// TwinCAT 3 PLC project Base
// ProgramVersion: 3.1.4022.4
// libraries:
//   Tc2_Standard, * (Beckhoff Automation GmbH)
//   Tc2_System, * (Beckhoff Automation GmbH)
//   Tc2_Utilities, * (Beckhoff Automation GmbH)
//   Tc3_IotBase, * (Beckhoff Automation GmbH)
//   Tc3_IotCommunicator, * (Beckhoff Automation GmbH)
//   Tc3_JsonXml, * (Beckhoff Automation GmbH)
//   Tc3_Module, * (Beckhoff Automation GmbH)
// project tree:
//   DUTs/ E_JsonStates.TcDUT (not stored), ST_ReceivedData.TcDUT
//   GVLs/ CELL_STATE.TcGVL (not stored), CELL_WORKING_STATES.TcGVL, CLAMP_STATE.TcGVL, CELL_ACTION_STATE.TcGVL (not stored), DATA_SERVICE_STATE.TcGVL (not stored), MHS_STATE.TcGVL (not stored), MHS_Registers.TcGVL
//   / PlcTask.TcTTO
//   POUs/ FB_Bool_To_Word.TcPOU (not stored), FB_Cell_Simu.TcPOU, FB_InterfaceProfibus.TcPOU (not stored), FB_RESTapi.TcPOU, FB_VirtualCell.TcPOU (not stored), FB_Word_To_Bool.TcPOU (not stored), I_CELL.TcIO, FB_Cell.TcPOU, FB_Clamp.TcPOU, FB_ClampSimulated.TcPOU, FB_DataService.TcPOU (not stored), FB_InterfaceIO.TcPOU (not stored), FB_InterfaceSimulated.TcPOU, FB_MHS.TcPOU, ITF_Cell.TcIO (not stored), JsonSaxHandler.TcPOU (not stored), MAIN.TcPOU, FB_VirtualCellIntWriter.TcPOU (not stored)
//   POUs/REST/ MAIN_1.TcPOU
//   POUs/REST/Postman/ FB_Get.TcPOU, FB_PUT.TcPOU
// real-time tasks:
//   TASK PlcTask: cycle T#10ms, priority 20, ADS port 350
// I/O:
//   DEVICE Device 3 (EtherCAT) (disabled), AmsNetId 192.168.74.113.4.1
//     Box 1 (CU1128) [CU1128 6x EtherCAT junction]
//       A2_Schaltschrank [EK1100 EtherCAT Coupler (2A E-Bus)]
//         Term 3 (EL2004) [EL2004 4Ch. Dig. Output 24V, 0.5A]
//         Term 4 (EL1004) [EL1004 4Ch. Dig. Input 24V, 3ms]
//         Term 5 (EL2004) [EL2004 4Ch. Dig. Output 24V, 0.5A]
//         Term 6 (EL2004) [EL2004 4Ch. Dig. Output 24V, 0.5A]
//         Term 7 (EL1004) [EL1004 4Ch. Dig. Input 24V, 3ms]
//         Term 8 (EL1004) [EL1004 4Ch. Dig. Input 24V, 3ms]
//         Term 9 (EL2004) [EL2004 4Ch. Dig. Output 24V, 0.5A]
//         Term 10 (EL1004) [EL1004 4Ch. Dig. Input 24V, 3ms]
//         Term 24 (EL9011) [EL9011 End Terminal]
//       A5 [EK1100 EtherCAT Coupler (2A E-Bus)]
//         Term 12 (EL1004) [EL1004 4Ch. Dig. Input 24V, 3ms]
//         Term 13 (EL1004) [EL1004 4Ch. Dig. Input 24V, 3ms]
//         Term 14 (EL2004) [EL2004 4Ch. Dig. Output 24V, 0.5A]
//         Term 15 (EL2004) [EL2004 4Ch. Dig. Output 24V, 0.5A]
//         Term 16 (EL2004) [EL2004 4Ch. Dig. Output 24V, 0.5A]
//         Term 25 (EL9011) [EL9011 End Terminal]
//       Dummy term [CU1128 6x EtherCAT junction - Dev A]
//         Term 18 (EK1100) [EK1100 EtherCAT Coupler (2A E-Bus)]
//           Term 19 (EL1004) [EL1004 4Ch. Dig. Input 24V, 3ms]
//           Term 20 (EL9505) [EL9505 Power supply terminal 5V]
//           Term 21 (EL1124) [EL1124 4Ch. Dig. Input 5V, 10µs, Sensor Power]
//           Term 22 (EL2124) [EL2124 4Ch. Dig. Output 5V, 20mA]
//           Term 26 (EL9011) [EL9011 End Terminal]
//       Term 25 (CU1128-C) [CU1128 6x EtherCAT junction - Dev B]

CONFIGURATION Base
    RESOURCE PLC ON TwinCAT3
        TASK PlcTask(INTERVAL := T#10ms, PRIORITY := 20);
        PROGRAM MAIN_1 WITH PlcTask : MAIN_1;
    END_RESOURCE
END_CONFIGURATION

// ---- DUTs/ST_ReceivedData.TcDUT
TYPE ST_ReceivedData :
STRUCT
	userId:	DINT;
	id:		DINT;
	title:	STRING(255);
	body:	STRING(255);
END_STRUCT
END_TYPE

// ---- GVLs/CELL_WORKING_STATES.TcGVL
{attribute 'qualified_only'}
VAR_GLOBAL
TYPE
	CELL_WORKING_STATES: (e_START, e_WORKING, e_DATAPUT,e_FINISHED);
END_TYPE		

END_VAR

// ---- GVLs/CLAMP_STATE.TcGVL
{attribute 'qualified_only'}
VAR_GLOBAL
TYPE
	CLAMP_STATE: (e_OPEN, e_CLOSED_FULL, e_CLOSED, e_ERROR);
END_TYPE		

END_VAR

// ---- GVLs/MHS_Registers.TcGVL
{attribute 'qualified_only'}
VAR_GLOBAL
 MHS : ARRAY [1..20] OF DINT;
END_VAR

// ---- POUs/I_CELL.TcIO
INTERFACE I_CELL

METHOD GetErrorString : STRING
VAR_INPUT
END_VAR
END_METHOD

METHOD GetName : STRING
VAR_INPUT
END_VAR
END_METHOD

METHOD GetState : INT
VAR_INPUT
END_VAR
END_METHOD

METHOD GetWorkpiece : DINT
VAR_INPUT
END_VAR
END_METHOD

METHOD IsDisassemblyCell : BOOL
VAR_INPUT
END_VAR
END_METHOD

METHOD IsError : BOOL
VAR_INPUT
END_VAR
END_METHOD

METHOD IsIdle : BOOL
VAR_INPUT
END_VAR
END_METHOD

METHOD IsVirtualCell : BOOL
VAR_INPUT
END_VAR
END_METHOD

METHOD RequestActionState : BOOL
VAR_INPUT
	csStateRequest : CELL_ACTION_STATE;
END_VAR
END_METHOD

METHOD RequestWork : BOOL
VAR_INPUT
END_VAR
END_METHOD

METHOD SetDisassemblyCell : BOOL
VAR_INPUT
	bIsDisassemblyCell : BOOL;
END_VAR
END_METHOD

METHOD SetGetDataServiceEnable : BOOL
VAR_INPUT
END_VAR
END_METHOD

METHOD SetName : BOOL
VAR_INPUT
	sName :string ;
END_VAR
END_METHOD

METHOD SetPutDataServiceEnable : BOOL
VAR_INPUT
END_VAR
END_METHOD

METHOD SetVirtualCell : BOOL
VAR_INPUT
END_VAR
END_METHOD

METHOD SetWorkpiece : BOOL
VAR_INPUT
	iWorkpiece : DINT;
	sWorkpieceID : STRING;
END_VAR
END_METHOD

METHOD StateMachine : BOOL
VAR_INPUT
END_VAR
END_METHOD

METHOD StateMachineProfibus : BOOL
VAR_INPUT
END_VAR
END_METHOD

END_INTERFACE

// ---- POUs/REST/MAIN_1.TcPOU
PROGRAM MAIN_1
VAR
	// trigger command execution for Postman-Echo samples
	
	
	fbMHS :  FB_MHS ;
	
	
	
	
END_VAR

fbMHS();

END_PROGRAM

// ---- POUs/FB_MHS.TcPOU
FUNCTION_BLOCK FB_MHS


VAR
	m_csStateRequest : MHS_STATE;
	m_csStateRequestOld : MHS_STATE;
	m_csState : MHS_STATE;
	m_csStateLastCycle : MHS_STATE;
	m_csStateLastAction : MHS_STATE;
	m_Name : STRING;	
	// Von SystemDemonstratorApp kommend
	m_iWorkpiece : DINT; 
	m_iCell : DINT;
	m_iRequest: DINT;
	// Von SystemDemonstratorApp kommend angenommen
	m_iWorkpieceAccepted : DINT; 
	m_iCellAccepted : DINT;
	m_iRequestAccepted: DINT;
	
	// Von PLC kommend 
	m_iMachineFree : DINT;	
	
	
	//Von MiR kommend
	m_iRequestMachineFree : DINT;
	m_iActionTerminated : DINT;	
	
	
	
	// Zustand der Zelle die Beladen oder Entladen werden soll
	m_eCurrentCellState : CELL_ACTION_STATE;
	m_eNeededCellState : CELL_ACTION_STATE;
	m_bNeededCellStatePending : BOOL;
	
	aMHS : ARRAY [1..20] OF DINT; // Interface API-Array
	
	
	m_iSimulationsTimer : DINT;
	
	///////////////////////////////////////////////////////////////////////////
	
	bGet, bPut   	: BOOL;
	

	
	fbClient				:  FB_IotHttpClient :=(sHostName:='jsonplaceholder.typicode.com',
								  	bKeepAlive:=TRUE, tConnectionTimeout:=T#10S);
								
	fbGet						:ARRAY [1..10] OF FB_Get;
	fbPut						:ARRAY [11..20] OF FB_PUT; 
	/////////////////////////////////////////////////////////////////////////////
	//*Hami* String Replace for URi
	
	s_URI : STRING  			:= '/posts/xx';
	i_Register	  				: INT ;
	s_i_Register				: STRING;
	S_Register_URi				: STRING;
	I							: INT ;
	i_I							: INT;
END_VAR

StateMachine();
//FOR i_Register:=1 TO 10  DO
//	i_Register := i_Register + 1;
//	s_i_Register := INT_TO_STRING(i_Register);
//	S_Register_URi := REPLACE(s_URI , s_i_Register , 2 , 8 );
	
//	I := I +1;
	
// END_FOR 

//IF NOT fbClient.bConfigured THEN 
//		fbClient.nHostPort:= 80;
//	END_IF 


/////////////////////////////////////////////////////////////////////////////////////////		

IF fbClient.bConfigured THEN 
		fbGet[1](bSend:=bGet,sURi := '/posts/1', fbClient:=fbClient);
		fbPut[11](bSend:=bPut,sURi := '/posts/1', fbClient:=fbClient);
END_IF

/////////////////////////////////////////////////////////////////////////////////////////		

IF fbClient.bConfigured THEN 
		fbGet[2](bSend:=bGet,sURi := '/posts/2', fbClient:=fbClient);
		fbPut[12](bSend:=bPut,sURi := '/posts/2', fbClient:=fbClient);
END_IF

/////////////////////////////////////////////////////////////////////////////////////////		

IF fbClient.bConfigured THEN 
		fbGet[3](bSend:=bGet,sURi := '/posts/3', fbClient:=fbClient);
		fbPut[13](bSend:=bPut,sURi := '/posts/3', fbClient:=fbClient);
END_IF

/////////////////////////////////////////////////////////////////////////////////////////		

IF fbClient.bConfigured THEN 
		fbGet[4](bSend:=bGet,sURi := '/posts/4', fbClient:=fbClient);
		fbPut[14](bSend:=bPut,sURi := '/posts/4', fbClient:=fbClient);
END_IF
/////////////////////////////////////////////////////////////////////////////////////////		

IF fbClient.bConfigured THEN 
		fbGet[5](bSend:=bGet,sURi := '/posts/5', fbClient:=fbClient);
		fbPut[15](bSend:=bPut,sURi := '/posts/5', fbClient:=fbClient);
END_IF


	fbClient.Execute();
	

	///////////////////////////// init client parameters at startup////////////////////////////////////
	
	

///////////////////////// SET MHS Connection///////////////////////////
// init client parameters at startup

/////////////////////////////////////////////////////////////////////
(*aMHS[1] := fbGet[1].q_iRegister;
aMHS[2] := fbGet[2].q_iRegister;
aMHS[3] := fbGet[3].q_iRegister;
aMHS[4] := fbGet[4].q_iRegister;
aMHS[5] := fbGet[5].q_iRegister;
aMHS[6] := fbGet[6].q_iRegister;
aMHS[7] := fbGet[7].q_iRegister;
aMHS[8] := fbGet[8].q_iRegister;
aMHS[9] := fbGet[9].q_iRegister;
aMHS[10] := fbGet[10].q_iRegister; 
*)

FOR I:=1 TO 10 DO
	aMHS[I] := fbGet[I].q_iRegister;
END_FOR


FOR i_I:=11 TO 20 DO
	fbPut[I].i_iRegister := aMHS[I];
END_FOR

METHOD GetActionFinished : BOOL
VAR_INPUT
END_VAR
IF m_csState = MHS_STATE.e_AKTION_FINISHED THEN
	GetActionFinished := TRUE;
ELSE
	GetActionFinished := FALSE;
END_IF
END_METHOD

METHOD GetCurrentCellForAction : DINT
VAR_INPUT
END_VAR
GetCurrentCellForAction := m_iCellAccepted;
END_METHOD

METHOD GetState : BOOL
VAR_INPUT
END_VAR
END_METHOD

METHOD NeededCellStatePending : BOOL
VAR_INPUT
END_VAR
NeededCellStatePending := m_bNeededCellStatePending;
m_bNeededCellStatePending := FALSE;
END_METHOD

METHOD RequestAction : BOOL
VAR_INPUT
	
	iWorkpiece : DINT; 
	iCell : DINT;
	bRequest : DINT;
END_VAR

m_iWorkpiece :=  iWorkpiece;
m_iCell := iCell;
m_iRequest := bRequest;
END_METHOD

METHOD RequestState : BOOL
VAR_INPUT
END_VAR
END_METHOD

METHOD SendNeededToCell : CELL_ACTION_STATE
VAR_INPUT
END_VAR
SendNeededToCell := m_eNeededCellState;
END_METHOD

METHOD SetClampIsOpen : BOOL
VAR_INPUT
iClampIsOpen : DINT;	

END_VAR
//IF iClampIsOpen > 0 THEN
//	m_iClampIsOpen := 1;
//	m_iClampIsClose := 0;
//ELSE
//	m_iClampIsOpen := 0;
//	m_iClampIsClose := 1;	
//END_IF
END_METHOD

METHOD SetDoorIsOpen : BOOL
VAR_INPUT
	iDoorIsOpen :DINT;
END_VAR
//IF iDoorIsOpen > 0 THEN
//	m_iDoorIsOpen := 1;
//	m_iDoorIsClose := 0;
//ELSE
//	m_iDoorIsOpen := 0;
//	m_iDoorIsClose := 1;	
//END_IF
END_METHOD

METHOD SetMachineFree : BOOL
VAR_INPUT
	iMachineFree:DINT;
END_VAR
m_iMachineFree := iMachineFree;
END_METHOD

METHOD SetStateCurrentMachineForAction : BOOL
VAR_INPUT
	eCurrentCellState :CELL_ACTION_STATE;
END_VAR
m_eCurrentCellState := eCurrentCellState;

SetStateCurrentMachineForAction := TRUE;
END_METHOD


METHOD StateMachine : BOOL
VAR_INPUT
END_VAR

VAR

END_VAR

	// VOM MHS

	//{define Simulated}
	{define MHSConnected}
	
	{IF defined (MHSConnected)}
 	m_iRequestMachineFree   := aMHS[11];
	m_iActionTerminated :=  aMHS[12];
	{END_IF}
	// PLC interne Variablen
	//m_iDoorIsOpen : DINT;	
	//m_iClampIsOpen : DINT;
	//m_iClampIsClose : DINT;	
	//m_iDoorIsClose : DINT;


	
	
CASE m_csState OF

MHS_STATE.e_IDLE: 

	IF m_iWorkpiece > 0 AND m_iCell > 0 AND m_iRequest > 0 THEN
		m_iWorkpieceAccepted := m_iWorkpiece;  
		m_iCellAccepted := m_iCell;
		m_iRequestAccepted:= m_iRequest; 	
	END_IF

	IF m_iWorkpieceAccepted > 0 AND m_iCellAccepted > 0 AND m_iRequestAccepted = 2 THEN
		aMHS[1] := m_iWorkpieceAccepted;
		aMHS[2] := m_iCellAccepted;
		aMHS[3] := m_iRequestAccepted;
		m_iWorkpiece := 0;
 		m_iCell := 0;
		m_iRequest := 0;
		m_csState := MHS_STATE.e_PGO_POS;	
	END_IF
	IF m_iWorkpieceAccepted > 0 AND m_iCellAccepted > 0 AND m_iRequestAccepted = 1 THEN
		aMHS[1] := m_iWorkpieceAccepted;
		aMHS[2] := m_iCellAccepted;
		aMHS[3] := m_iRequestAccepted;
		m_iWorkpiece := 0;
 		m_iCell := 0;
		m_iRequest := 0;
		m_csState := MHS_STATE.e_GGO_POS;	
	END_IF
	// Löschen dieser Anforderung
	m_iRequestAccepted := 0;


// SUBROUTINE WP in Maschine bringen	  
MHS_STATE.e_PGO_POS:
	
 	IF m_iRequestMachineFree > 0 THEN
		m_eNeededCellState := CELL_ACTION_STATE.e_LoadPos;
		m_bNeededCellStatePending := TRUE;
		m_csState := MHS_STATE.e_PWAIT_DOOR;
	END_IF
	

MHS_STATE.e_PWAIT_DOOR:	
  	IF  m_eCurrentCellState = CELL_ACTION_STATE.e_LoadPos THEN
		//aMHS[3] := 0;//m_iRequest;
		m_iMachineFree := 1;
		m_csState := MHS_STATE.e_PWAIT_CLAMP;
	END_IF

MHS_STATE.e_PWAIT_CLAMP:
		m_csState := MHS_STATE.e_PPUT_WP;
	

MHS_STATE.e_PPUT_WP:
		m_csState := MHS_STATE.e_PCLOSE_CLAMP;
		
 MHS_STATE.e_PCLOSE_CLAMP:
			m_csState := MHS_STATE.e_PLEAFE_MACHINE;
	 
MHS_STATE.e_PLEAFE_MACHINE:
 	IF m_iActionTerminated > 0 THEN
		m_csState := MHS_STATE.e_AKTION_FINISHED;
	END_IF	

// SUBROUTINE WP aus Maschine holen	  
MHS_STATE.e_GGO_POS:
 	IF m_iRequestMachineFree > 0 THEN
		m_eNeededCellState := CELL_ACTION_STATE.e_UnLoadPos;
		m_bNeededCellStatePending := TRUE;
		m_csState := MHS_STATE.e_GWAIT_DOOR;
	END_IF

	
MHS_STATE.e_GWAIT_DOOR:
  	IF  m_eCurrentCellState = CELL_ACTION_STATE.e_UnLoadPos THEN
		m_iMachineFree := 1;
		//aMHS[3] := 0;//m_iRequest;
		m_csState := MHS_STATE.e_GWAIT_CLAMP;
	END_IF

MHS_STATE.e_GWAIT_CLAMP:
	//IF m_iClampIsOpen > 0 THEN
		m_csState := MHS_STATE.e_GGET_WP;
	//END_IF
MHS_STATE.e_GGET_WP:
	//IF 	m_iClampCloseRequest > 0 THEN
		m_csState := MHS_STATE.e_GCLOSE_CLAMP;
	//END_IF
 MHS_STATE.e_GCLOSE_CLAMP:
 	//IF m_iClampIsClose > 0 THEN
			m_csState := MHS_STATE.e_GLEAFE_MACHINE;	 
 	//END_IF
MHS_STATE.e_GLEAFE_MACHINE:
	
 	IF m_iActionTerminated > 0 THEN
		aMHS[3] := 0;//m_iRequest;
		m_csState := MHS_STATE.e_AKTION_FINISHED;
	END_IF		

MHS_STATE.e_AKTION_FINISHED:
	m_csState := MHS_STATE.e_IDLE;
	m_iMachineFree := 0;
	
MHS_STATE.e_ERROR:
	
ELSE
	m_csState := MHS_STATE.e_ERROR;
 
END_CASE
{IF defined (MHSConnected)}
aMHS[4] :=  m_iMachineFree; 
{END_IF}
END_METHOD

END_FUNCTION_BLOCK

// ---- POUs/REST/Postman/FB_Get.TcPOU
FUNCTION_BLOCK FB_Get
VAR_INPUT
	bSend				: BOOL;
	sURi : STRING;
	
END_VAR
VAR_IN_OUT
	fbClient			: FB_IotHttpClient;
END_VAR
VAR_OUTPUT
	bBusy				: BOOL;
	bError				: BOOL;
	q_iRegister 		: DINT;
END_VAR
VAR
	fbHeader: FB_IotHttpHeaderFieldMap ;
	fbRequest			: FB_IotHttpRequest;
	fbJson				: FB_JsonDomParser;
	nState				: UDINT;
	RisingEdge			: R_TRIG;
	
	bGetContentResult	: BOOL;
	sContent			: STRING(511);
	
	bGetJsonResult		: BOOL;
	jsonDoc				: SJsonValue;
	jsonVal				: SJsonValue;
	newJSONval : SJsonValue;
	sResultValue		: STRING;
	
	nReqCount			: UDINT;	
	nResCount			: UDINT;
	nValidResCount		: UDINT;
	nErrCount			: UDINT;
	b : BOOL ;
	stReceivedData : ST_ReceivedData ;
	bOnce: BOOL;
	
END_VAR

 IF bOnce THEN
	fbHeader.AddField('Authorization', 'Basic RmVsaXg6OGM2OTc2ZTViNTQxMDQxNWJkZTkwOGJkNGRlZTE1ZGZiMTY3YTljODczZmM0YmI4YTgxZjZmMmFiNDQ4YTkxOA==', FALSE);
	fbHeader.AddField('Accept-Language', 'de_DE' , FALSE);
	bOnce:= FALSE;
END_IF


RisingEdge(CLK:= bSend );
CASE nState OF
0:	
	IF RisingEdge.Q THEN 
		IF fbRequest.SendRequest(sURi:=sURi, fbClient:=fbClient, eRequestType:=ETcIotHttpRequestType.HTTP_GET, 0, 0, 0) THEN	
//IF fbRequest.GetJsonDomContent(sURi := '/posts/1/' , fbClient := fbClient , eRequestType:=ETcIotHttpRequestType.HTTP_GET ,fbJson := fbJson,0) THEN				
			nState:= 1;
			nReqCount:= nReqCount+1;
			bBusy:= TRUE;
			bError:= FALSE;
		END_IF					
	END_IF
1:
	IF NOT fbRequest.bBusy THEN
		bError:= TRUE;
		IF NOT fbRequest.bError THEN
				bGetContentResult:= fbRequest.GetContent(pContent:= ADR(sContent), nContentSize:= SIZEOF(sContent), bSetNullTermination:= TRUE);
			IF fbRequest.nStatusCode >= 200 AND fbRequest.nStatusCode < 300 THEN
				bGetJsonResult:= FALSE;
				jsonDoc:= fbRequest.GetJsonDomContent(fbJson);
				IF jsonDoc <> 0 THEN
					bGetJsonResult:= TRUE;
					IF fbJson.HasMember(jsonDoc, 'id')  THEN
						jsonVal:= fbJson.FindMember(jsonDoc, 'id');
						q_iRegister := fbJson.GetInt(jsonVal);
						IF fbJson.HasMember(jsonVal, 'title')  THEN
							jsonVal:= fbJson.FindMember(jsonVal, 'title');
							nValidResCount:= nValidResCount+1;
							bError:= FALSE;						
							IF fbJson.IsString(jsonVal) THEN							
								sResultValue:= fbJson.GetString(jsonVal);									
							END_IF
						END_IF		
					END_IF
				END_IF							
				nResCount:= nResCount+1;			
			END_IF
		END_IF
		nState:= 0;
		bBusy:= FALSE;
		IF bError THEN
			nErrCount:= nErrCount+1;
		END_IF
	END_IF  	
END_CASE

END_FUNCTION_BLOCK

// ---- POUs/REST/Postman/FB_PUT.TcPOU
FUNCTION_BLOCK FB_PUT
VAR_INPUT
	bSend		: BOOL;
	i_iRegister : DINT ;
	sURi 		: STRING;
END_VAR
VAR_IN_OUT
	fbClient			: FB_IotHttpClient;
END_VAR
VAR_OUTPUT
	bBusy				: BOOL;
	bError				: BOOL;
END_VAR
VAR
	fbRequest			: FB_IotHttpRequest;
	fbHeader			: FB_IotHttpHeaderFieldMap;
	fbJson				: FB_JsonDomParser;
	//fbJson			: FB_JsonDomParser;
	nState				: UDINT;
	RisingEdge			: R_TRIG;

	bGetContentResult	: BOOL;
	sContent			: STRING(511);
	
	bGetJsonResult		: BOOL;
	jsonDoc				: SJsonValue;
	jsonVal				: SJsonValue;
	bResultValue		: BOOL;
	
	nReqCount			: UDINT;	
	nResCount			: UDINT;
	nValidResCount		: UDINT;
	nErrCount			: UDINT;
	bOnce				: BOOL:= TRUE;
	l_sMessage 			: STRING(255) := '{"id":"5","title":"1547mV"}';
	sMessage			: STRING(255);
	JsonStringValue		: SJsonValue;
	s_iRegister 		: STRING ;
	ss_iRegister		: STRING ;
END_VAR

IF bOnce THEN
	fbHeader.AddField('Authorization', 'Basic RmVsaXg6OGM2OTc2ZTViNTQxMDQxNWJkZTkwOGJkNGRlZTE1ZGZiMTY3YTljODczZmM0YmI4YTgxZjZmMmFiNDQ4YTkxOA==', FALSE);
	fbHeader.AddField('Accept-Language', 'de_DE' , FALSE);
	bOnce:= FALSE;
END_IF

/////////////////////////////////////////////////////////////////////////////
s_iRegister := DINT_TO_STRING(i_iRegister);
sMessage := REPLACE(l_sMessage,s_iRegister,1,8);
JsonStringValue := fbJson.ParseDocument(sMessage);

/////////////////////////////////////////////////////////////////////////////
RisingEdge(CLK:= bSend);
CASE nState OF
0:	
	IF RisingEdge.Q THEN 
		IF fbRequest.SendJsonDomRequest(sUri:= sURi , fbClient:=fbClient, eRequestType:=ETcIotHttpRequestType.HTTP_PUT, fbJson := fbJson, fbHeader:=fbHeader) THEN				
			nState:= 1;
			nReqCount:= nReqCount+1;
			bBusy:= TRUE;
			bError:= FALSE;
		END_IF					
	END_IF
1:
	IF NOT fbRequest.bBusy THEN
		bError:= TRUE;
		IF NOT fbRequest.bError THEN				 
			bGetContentResult:= fbRequest.GetContent(pContent:= ADR(sContent), nContentSize:= SIZEOF(sContent), bSetNullTermination:= TRUE);
			IF fbRequest.nStatusCode >= 200 AND fbRequest.nStatusCode < 300 THEN
				bGetJsonResult:= FALSE;
				jsonDoc:= fbRequest.GetJsonDomContent(fbJson);
				IF jsonDoc <> 0 THEN
					bGetJsonResult:= TRUE;
					
					IF fbJson.HasMember(jsonDoc, 'id') THEN
					//IF fbJson.HasMember(jsonDoc, 'authenticated') THEN
					jsonVal:= fbJson.FindMember(jsonDoc, 'id');
						//jsonVal:= fbJson.FindMember(jsonDoc, 'authenticated');
						IF fbJson.IsInt(jsonVal) THEN
						//IF fbJson.IsBool(jsonVal) THEN
						i_iRegister:= fbJson.GetInt(jsonVal);
							//bResultValue:= fbJson.GetBool(jsonVal);
							nValidResCount:= nValidResCount+1;
							bError:= FALSE;						
						END_IF	
					END_IF
				END_IF							
				nResCount:= nResCount+1;			
			END_IF
		END_IF
		nState:= 0;
		bBusy:= FALSE;
		IF bError THEN
			nErrCount:= nErrCount+1;
		END_IF
	END_IF  	
END_CASE

END_FUNCTION_BLOCK

// ---- POUs/FB_Cell_Simu.TcPOU
FUNCTION_BLOCK FB_Cell_Simu IMPLEMENTS I_CELL
VAR_INPUT
	
END_VAR
VAR_OUTPUT
END_VAR
VAR
	m_csStateRequest : CELL_ACTION_STATE;
	m_csStateRequestOld : CELL_ACTION_STATE;
	m_csState : CELL_ACTION_STATE;
	m_csStateLastCycle : CELL_ACTION_STATE;
	m_csStateLastAction : CELL_ACTION_STATE;
	
	
	m_csSRWorkingState : CELL_WORKING_STATES := CELL_WORKING_STATES.e_FINISHED;
	m_csSRWorkingStateLast : CELL_WORKING_STATES := CELL_WORKING_STATES.e_FINISHED;
	// Eigenschaften
	m_sName : STRING;
	m_bIsDisassemblyCell : BOOL;
	
	
	m_iWorkpiece : DINT;
	m_sWorkpieceID : STRING;
	

	m_csCellState : CELL_STATE;
	m_csCellStateLast : CELL_STATE;

	fbInterface : FB_InterfaceSimulated; //nn wenn keine Eingeänge vorhanden sind, nach zeiten wechsel
	fbClamp : FB_Clamp; 
	
	m_sErrorString : STRING;
	
	// DataServices
	
	fbDataServicePut : FB_DataService;
	m_bDataServicePutEnable : BOOL;
	fbDataServiceGet : FB_DataService;
	m_bDataServiceGetEnable : BOOL;
	m_sConfigString : STRING;
	m_sConfigStringEndGet : STRING  := '_Get.exe';
	m_sConfigStringEndPut : STRING  := '_Put.exe';
	m_sDataServiceDir: STRING  := 'C:\Users\\Nübel\Desktop\Sysdem_Nü_Ulitmate\CUTS\';
	m_sDataServiceIP: STRING  := '192.168.74.113.1.1';
	
END_VAR

METHOD GetErrorString : STRING
VAR_INPUT
END_VAR
END_METHOD

METHOD GetName : STRING
VAR_INPUT
END_VAR
GetName := m_sName;
END_METHOD

METHOD PUBLIC GetState : INT
VAR_INPUT
	
END_VAR
GetState := m_csState;
END_METHOD

METHOD GetWorkpiece : DINT
VAR_INPUT
END_VAR
GetWorkpiece := m_iWorkpiece;
END_METHOD

METHOD IsDisassemblyCell : BOOL
VAR_INPUT
END_VAR
IsDisassemblyCell := m_bIsDisassemblyCell;
END_METHOD

METHOD IsError : BOOL
VAR_INPUT
END_VAR
IF m_csCellState = CELL_STATE.e_ERROR THEN
	IsError := TRUE;
END_IF
END_METHOD

METHOD IsIdle : BOOL
VAR_INPUT
END_VAR
IF m_csCellState = CELL_STATE.e_IDEL THEN
	IsIdle := TRUE;
END_IF
END_METHOD

METHOD IsVirtualCell : BOOL
VAR_INPUT
END_VAR
IsVirtualCell :=FALSE;
END_METHOD

METHOD PUBLIC RequestActionState : BOOL
VAR_INPUT
	csStateRequest : CELL_ACTION_STATE;
END_VAR
m_csStateRequest := csStateRequest;
END_METHOD

METHOD RequestWork : BOOL
VAR_INPUT
END_VAR
m_csCellState := CELL_STATE.e_WORKING;
END_METHOD

METHOD SetDisassemblyCell : BOOL
VAR_INPUT
	bIsDisassemblyCell : BOOL;
END_VAR
m_bIsDisassemblyCell := bIsDisassemblyCell;
END_METHOD

METHOD SetGetDataServiceEnable : BOOL
VAR_INPUT
END_VAR
m_bDataServiceGetEnable := TRUE;
SetGetDataServiceEnable := TRUE;
END_METHOD

METHOD SetName : BOOL
VAR_INPUT
	sName :string ;
END_VAR
m_sName := sName;
END_METHOD

METHOD SetPutDataServiceEnable : BOOL
VAR_INPUT
END_VAR
m_bDataServicePutEnable := TRUE;
SetPutDataServiceEnable := TRUE;
END_METHOD

METHOD SetVirtualCell : BOOL
VAR_INPUT
END_VAR
END_METHOD

METHOD SetWorkpiece : BOOL
VAR_INPUT
	iWorkpiece : DINT;
	sWorkpieceID : STRING;
END_VAR
m_iWorkpiece := iWorkpiece;
m_sWorkpieceID := sWorkpieceID;
END_METHOD

METHOD PUBLIC StateMachine : BOOL
VAR_INPUT
END_VAR

fbInterface();
fbClamp();



// Error-Abfragen
IF fbClamp.IsError() THEN
	m_csCellState := CELL_STATE.e_ERROR; 
	m_sErrorString := 'CLAMP-Error: Clamp is closed without Workpiece';
END_IF


//Zellen Zustandsmaschine

CASE m_csCellState OF 
	CELL_STATE.e_IDEL:
		fbClamp.SetOpenClamp();	
	
		;
 	CELL_STATE.e_MHS_ACTION;
		//SubRoutine für Aktion beim beladen aktuell leer da alles vom MHS gesteuert wird 
	
		;
	CELL_STATE.e_WORKING:
		//SubRoutine zum Durchführen einer Bearbeitung
		
		IF NOT (m_csCellStateLast = m_csCellState) THEN
			m_csSRWorkingState := CELL_WORKING_STATES.e_START;
			IF m_bDataServiceGetEnable THEN
				fbDataServiceGet.SetNetIP('192.168.74.113.1.1');
				fbDataServiceGet.SetWorkingDirectory('C:\Users\Nübel\Desktop\Sysdem_Nü_Ulitmate\CUTS');
				m_sConfigString := 'C:\Users\Nübel\Desktop\Sysdem_Nü_Ulitmate\CUTS\';
				m_sConfigString := CONCAT(m_sConfigString , m_sName); // erstellen des Pfades der Applikation 
				m_sConfigString := CONCAT(m_sConfigString , m_sConfigStringEndGet);
				fbDataServiceGet.SetCommandLine(m_sWorkpieceID);
				fbDataServiceGet.SetPathOfApplication(m_sConfigString);
				fbDataServiceGet.StartDataService();
			END_IF
		END_IF
			
		CASE m_csSRWorkingState OF
			
			CELL_WORKING_STATES.e_START:
				
				IF NOT (m_csSRWorkingStateLast = m_csSRWorkingState )THEN
					m_csStateRequest := CELL_ACTION_STATE.e_Startabel;
				END_IF
				//m_csSRWorkingState:= CELL_WORKING_STATES.e_FINISHED;
				
				IF m_csState = CELL_ACTION_STATE.e_Startabel AND (fbDataServiceGet.IsFinished() OR NOT(m_bDataServiceGetEnable) )  THEN // Zelle bereit zum Starten und DataServiceGet fertig oder nicht konfiguriert
					m_csSRWorkingState:= CELL_WORKING_STATES.e_WORKING;
					fbDataServiceGet.SetIdle();
					m_csStateRequest:= CELL_ACTION_STATE.e_Running;
				END_IF
				
				
			CELL_WORKING_STATES.e_WORKING:
				IF NOT (m_csSRWorkingStateLast = m_csSRWorkingState) THEN
					m_csStateRequest := CELL_ACTION_STATE.e_Running;
				END_IF
				
				IF m_csState = CELL_ACTION_STATE.e_Finished THEN
					m_csSRWorkingState := CELL_WORKING_STATES.e_FINISHED;
					IF m_bDataServicePutEnable THEN
						fbDataServicePut.SetNetIP('192.168.74.113.1.1');
						fbDataServicePut.SetWorkingDirectory('C:\Users\Nübel\Desktop\Sysdem_Nü_Ulitmate\CUTS');
						m_sConfigString := 'C:\Users\Nübel\Desktop\Sysdem_Nü_Ulitmate\CUTS\';						
						m_sConfigString := CONCAT(m_sConfigString , m_sName); // erstellen des Pfades der Applikation 
						m_sConfigString := CONCAT(m_sConfigString , m_sConfigStringEndPut);// erstellen des Pfades der Applikation
						fbDataServicePut.SetCommandLine(m_sWorkpieceID);
						fbDataServicePut.SetPathOfApplication(m_sConfigString);
						fbDataServicePut.StartDataService();
						m_csSRWorkingState := e_DATAPUT;
					END_IF
		
				END_IF
			CELL_WORKING_STATES.e_DATAPUT:
				
					IF fbDataServicePut.IsFinished() THEN
						fbDataServicePut.SetIdle();
						m_csSRWorkingState := CELL_WORKING_STATES.e_FINISHED;
					END_IF
					
					IF fbDataServicePut.IsError() THEN
						fbDataServicePut.SetIdle();
						m_csSRWorkingState := CELL_STATE.e_ERROR;
					END_IF
					
			CELL_WORKING_STATES.e_FINISHED:
				m_csCellState := CELL_STATE.e_IDEL;
			
		END_CASE		
		
	CELL_STATE.e_ERROR:
		m_csState :=CELL_ACTION_STATE.e_ToEmergencyStop;
	
		
END_CASE
m_csSRWorkingStateLast := m_csSRWorkingState;
m_csCellStateLast := m_csCellState;

IF NOT (m_csStateRequestOld = m_csStateRequest) THEN
	m_csState := m_csStateRequest - 1;
	m_csStateRequestOld := m_csStateRequest;
END_IF


// Aktions Zustandsmaschine
CASE m_csState OF 
	CELL_ACTION_STATE.e_ToStandby:
		IF NOT (m_csStateLastCycle = m_csState) THEN
			fbInterface.SetStandby(TRUE);
			m_csStateLastAction := m_csStateLastCycle;
		END_IF
		
		IF fbInterface.GetStandby() THEN
			m_csState := e_Standby; 
		END_IF
		
	CELL_ACTION_STATE.e_Standby :
	
		IF NOT (m_csStateLastCycle = m_csState) THEN
			m_csStateLastAction := m_csStateLastCycle;
		END_IF
		fbInterface.SetStandby(FALSE);
		
	CELL_ACTION_STATE.e_ToLoadPos:
	
		IF NOT (m_csStateLastCycle = m_csState) THEN
			m_csStateLastAction := m_csStateLastCycle;
			fbInterface.SetMoveToLoad(TRUE);
			fbClamp.SetOpenClamp();
		END_IF
		
		IF fbInterface.GetLoadPos() AND fbClamp.IsOpen() THEN
			m_csState := e_LoadPos; 
		END_IF
		
		
	CELL_ACTION_STATE.e_LoadPos:
	
		IF NOT (m_csStateLastCycle = m_csState) THEN
			m_csStateLastAction := m_csStateLastCycle;
		END_IF
		fbInterface.SetMoveToLoad(FALSE);
				
		
	CELL_ACTION_STATE.e_ToStartabel:
	
		IF NOT (m_csStateLastCycle = m_csState) THEN
			m_csStateLastAction := m_csStateLastCycle;
			fbClamp.SetCloseClampFull();
		END_IF
		
		
		IF  fbClamp.IsClosedFull() THEN
			m_csState := e_Startabel; 
		END_IF
		
	CELL_ACTION_STATE.e_Startabel:
	
		IF NOT (m_csStateLastCycle = m_csState) THEN
			m_csStateLastAction := m_csStateLastCycle;
			
		END_IF
		
	CELL_ACTION_STATE.e_ToRunning:
	
		IF NOT (m_csStateLastCycle = m_csState) THEN
			m_csStateLastAction := m_csStateLastCycle;
			fbInterface.SetStart(TRUE);
		END_IF
		
		IF fbInterface.GetIsRunning() THEN
			m_csState := CELL_ACTION_STATE.e_Running; 
		END_IF
		
	CELL_ACTION_STATE.e_Running:
	
		IF NOT (m_csStateLastCycle = m_csState) THEN
			m_csStateLastAction := m_csStateLastCycle;
		END_IF
		fbInterface.SetStart(FALSE);
		IF fbInterface.GetFinished() THEN
			m_csState := CELL_ACTION_STATE.e_Finished;		
		END_IF
	CELL_ACTION_STATE.e_Finished:
		IF NOT (m_csStateLastCycle = m_csState) THEN
			m_csStateLastAction := m_csStateLastCycle;
		END_IF
		
	CELL_ACTION_STATE.e_ToUnLoadPos:
 
		IF NOT (m_csStateLastCycle = m_csState) THEN
			m_csStateLastAction := m_csStateLastCycle;
			fbClamp.SetOpenClamp();
			fbInterface.SetMoveToUnload(TRUE);
			
		END_IF
		
		
		IF fbInterface.GetUnloadPos() AND fbClamp.IsOpen() THEN
			m_csState := e_UnLoadPos; 
			fbInterface.SetMoveToUnload(FALSE);
		END_IF
		
	CELL_ACTION_STATE.e_UnLoadPos:
	
		IF NOT (m_csStateLastCycle = m_csState) THEN
			m_csStateLastAction := m_csStateLastCycle;
		END_IF
		
	CELL_ACTION_STATE.e_ToEmergencyStop:
	
		IF NOT (m_csStateLastCycle = m_csState) THEN
			m_csStateLastAction := m_csStateLastCycle;
		END_IF
		
		
		IF fbInterface.GetEmergencyStop() THEN
			m_csState := e_EmergencyStop; 
		END_IF
		
	CELL_ACTION_STATE.e_EmergencyStop:
	
		IF NOT (m_csStateLastCycle = m_csState) THEN
			m_csStateLastAction := m_csStateLastCycle;
		END_IF
		
	CELL_ACTION_STATE.e_ToEmergencyOff:
	
		IF NOT (m_csStateLastCycle = m_csState) THEN
			m_csStateLastAction := m_csStateLastCycle;
		END_IF
		
		
		IF fbInterface.GetEmergencyStop() THEN
			m_csState := e_EmergencyOff; 
		END_IF
		
	CELL_ACTION_STATE.e_EmergencyOff:
	
		IF NOT (m_csStateLastCycle = m_csState) THEN
			m_csStateLastAction := m_csStateLastCycle;
		END_IF
		
	ELSE
		IF NOT (m_csStateLastCycle = m_csState) THEN
			m_csStateLastAction := m_csStateLastCycle;
		END_IF
		
END_CASE

IF m_bDataServiceGetEnable THEN
	fbDataServiceGet();
END_IF
IF m_bDataServicePutEnable THEN	
	fbDataServicePut();
END_IF

m_csStateLastCycle := m_csState;
END_METHOD

METHOD StateMachineProfibus : BOOL
VAR_INPUT
END_VAR
END_METHOD

END_FUNCTION_BLOCK

// ---- POUs/FB_InterfaceSimulated.TcPOU
FUNCTION_BLOCK FB_InterfaceSimulated IMPLEMENTS ITF_Cell
VAR_INPUT
END_VAR
VAR_OUTPUT
END_VAR
VAR
	 iTimer : INT;
	 iWaitingTime : INT := 500;
END_VAR

METHOD GetEmergencyOff : BOOL
VAR_INPUT
END_VAR

iTimer := iTimer +1;

IF iTimer > iWaitingTime THEN
	GetEmergencyOff := TRUE;
	iTimer := 0;	
END_IF
END_METHOD

METHOD GetEmergencyStop : BOOL
VAR_INPUT
END_VAR

iTimer := iTimer +1;

IF iTimer > iWaitingTime THEN
	GetEmergencyStop := TRUE;
	iTimer := 0;	
END_IF
END_METHOD

METHOD GetFinished : BOOL
VAR_INPUT
END_VAR

iTimer := iTimer +1;

IF iTimer > iWaitingTime THEN
	GetFinished := TRUE;
	iTimer := 0;	
END_IF
END_METHOD

METHOD GetIsRunning : BOOL
VAR_INPUT
END_VAR


iTimer := iTimer +1;

IF iTimer > iWaitingTime THEN
	GetIsRunning := TRUE;
	iTimer := 0;	
END_IF
END_METHOD

METHOD GetLoadPos : BOOL
VAR_INPUT
END_VAR


iTimer := iTimer +1;

IF iTimer > iWaitingTime THEN
	GetLoadPos := TRUE;
	iTimer := 0;	
END_IF
END_METHOD

METHOD GetStandby : BOOL
VAR_INPUT
END_VAR


iTimer := iTimer +1;

IF iTimer > iWaitingTime THEN
	GetStandby := TRUE;
	iTimer := 0;	
END_IF
END_METHOD

METHOD GetStartable : BOOL
VAR_INPUT
END_VAR



iTimer := iTimer +1;

IF iTimer > iWaitingTime THEN
	GetStartable := TRUE;
	iTimer := 0;	
END_IF
END_METHOD

METHOD GetUnloadPos : BOOL
VAR_INPUT
END_VAR


iTimer := iTimer +1;

IF iTimer > iWaitingTime THEN
	GetUnloadPos := TRUE;
	iTimer := 0;	
END_IF
END_METHOD

METHOD SetEmergencyOff : BOOL
VAR_INPUT
	b:BOOL;
END_VAR
END_METHOD

METHOD SetEmergencyStop : BOOL
VAR_INPUT
	b:BOOL;
END_VAR
END_METHOD

METHOD SetLoadPlace : BOOL
VAR_INPUT
	b :BOOL;
END_VAR
END_METHOD

METHOD SetMoveToLoad : BOOL
VAR_INPUT
	b:BOOL;
END_VAR
END_METHOD

METHOD SetMoveToUnload : BOOL
VAR_INPUT
	b:BOOL;
END_VAR
END_METHOD

METHOD SetStandby : BOOL
VAR_INPUT
	b:BOOL;
END_VAR
END_METHOD

METHOD SetStart : BOOL
VAR_INPUT
	b:BOOL;
END_VAR
END_METHOD

END_FUNCTION_BLOCK

// ---- POUs/FB_Clamp.TcPOU
FUNCTION_BLOCK FB_Clamp
VAR_INPUT
	
END_VAR
VAR_OUTPUT
END_VAR
VAR
m_csState : CLAMP_STATE;	
m_csStateRequested : CLAMP_STATE;

//Eingänge
m_bIsOpen AT %I* : BOOL;
m_bIsClosed AT %I* : BOOL;
m_bIsFull AT %I* : BOOL;

//Ausgänge
m_bOpen AT %Q* :BOOL;


END_VAR


StateMachine();

METHOD IsClosed : BOOL
VAR_INPUT
END_VAR
IF m_csState = CLAMP_STATE.e_CLOSED THEN
	IsClosed := TRUE;
END_IF
END_METHOD

METHOD IsClosedFull : BOOL
VAR_INPUT
END_VAR
IF m_csState = CLAMP_STATE.e_CLOSED_FULL THEN
	IsClosedFull := TRUE;
END_IF
END_METHOD

METHOD IsError : BOOL
VAR_INPUT
END_VAR
IF m_csState = CLAMP_STATE.e_ERROR THEN
	IsError := TRUE;
END_IF
END_METHOD

METHOD IsOpen : BOOL
VAR_INPUT
END_VAR
IF m_csState = CLAMP_STATE.e_OPEN THEN
	IsOpen := TRUE;
END_IF
END_METHOD

METHOD SetCloseClampEmpty : BOOL
VAR_INPUT
END_VAR
m_csStateRequested := CLAMP_STATE.e_CLOSED;
m_bOpen := FALSE;
SetCloseClampEmpty:=TRUE;
END_METHOD

METHOD SetCloseClampFull : BOOL
VAR_INPUT
END_VAR
m_csStateRequested := CLAMP_STATE.e_CLOSED_FULL;
m_bOpen := FALSE;
SetCloseClampFull := TRUE;
END_METHOD

METHOD SetOpenClamp : BOOL
VAR_INPUT
END_VAR
m_bOpen := TRUE;
END_METHOD

METHOD StateMachine : BOOL
VAR_INPUT
END_VAR

//m_bIsOpen : BOOL;
//m_bIsClosed : BOOL;
//m_bIsClosedFull : BOOL;

CASE m_csState  OF
	
	CLAMP_STATE.e_OPEN:	

		IF m_bIsClosed THEN
			IF 	m_bIsFull THEN
				m_csState := CLAMP_STATE.e_CLOSED_FULL;		
			ELSE
				m_csState := CLAMP_STATE.e_CLOSED;		
			END_IF 
		
		END_IF
		
		
 	CLAMP_STATE.e_CLOSED_FULL:
	// Fehler wenn falscher Zustand
 		IF m_csStateRequested = CLAMP_STATE.e_CLOSED THEN
  			m_csState := CLAMP_STATE.e_ERROR;
		END_IF
		
		
		IF m_bIsOpen THEN
			m_csState := CLAMP_STATE.e_OPEN;		
		END_IF
	
	CLAMP_STATE.e_CLOSED:
			// Fehler wenn falscher Zustand in diesem Fall: Werkstück erwartet aber nicht im Halter
 		IF m_csStateRequested = CLAMP_STATE.e_CLOSED_FULL THEN
  			m_csState := CLAMP_STATE.e_ERROR;
		END_IF
	
		IF m_bIsOpen THEN
			m_csState := CLAMP_STATE.e_OPEN;		
		END_IF
		
CLAMP_STATE.e_ERROR:
		
END_CASE
END_METHOD

END_FUNCTION_BLOCK

// ---- POUs/FB_RESTapi.TcPOU
FUNCTION_BLOCK FB_RESTapi
VAR_INPUT
END_VAR
VAR_OUTPUT
END_VAR
VAR
	fbREST : 
END_VAR

END_FUNCTION_BLOCK

// ---- POUs/FB_Cell.TcPOU
FUNCTION_BLOCK FB_Cell IMPLEMENTS I_CELL
VAR_INPUT
	
END_VAR
VAR_OUTPUT
END_VAR
VAR
	m_csStateRequest : CELL_ACTION_STATE;
	m_csStateRequestOld : CELL_ACTION_STATE;
	m_csState : CELL_ACTION_STATE;
	m_csStateLastCycle : CELL_ACTION_STATE;
	m_csStateLastAction : CELL_ACTION_STATE;
	
	
	m_csSRWorkingState : CELL_WORKING_STATES := CELL_WORKING_STATES.e_FINISHED;
	m_csSRWorkingStateLast : CELL_WORKING_STATES := CELL_WORKING_STATES.e_FINISHED;
	// Eigenschaften
	m_sName : STRING;
	m_bIsDisassemblyCell : BOOL;
	
	
	m_iWorkpiece : DINT;
	m_sWorkpieceID : STRING;
	

	m_csCellState : CELL_STATE;
	m_csCellStateLast : CELL_STATE;

	fbInterface : FB_InterfaceIO;
	//*Hami* Deklration von FB_InterfaceProfibus (Die Wurde in Method (StateMachine)) aufgerufen
	fbInterfaceProfibus : FB_InterfaceProfibus;
	fbClamp : FB_Clamp; 
	
	m_sErrorString : STRING;
	
	// DataServices
	
	fbDataServicePut : FB_DataService;
	m_bDataServicePutEnable : BOOL;
	fbDataServiceGet : FB_DataService;
	m_bDataServiceGetEnable : BOOL;
	m_sConfigString : STRING;
	m_sConfigStringEndGet : STRING  := '_Get.exe';
	m_sConfigStringEndPut : STRING  := '_Put.exe';

	m_sDataServiceDir: STRING  := 'C:\Users\\Nübel\Desktop\Sysdem_Nü_Ulitmate\CUTS\';
	m_sDataServiceIP: STRING  := '192.168.74.113.1.1';
	

	
	
END_VAR

METHOD GetErrorString : STRING
VAR_INPUT
END_VAR
END_METHOD

METHOD GetName : STRING
VAR_INPUT
END_VAR
GetName := m_sName;
END_METHOD

METHOD PUBLIC GetState : INT
VAR_INPUT
	
END_VAR
GetState := m_csState;
END_METHOD

METHOD GetWorkpiece : DINT
VAR_INPUT
END_VAR
GetWorkpiece := m_iWorkpiece;
END_METHOD

METHOD IsDisassemblyCell : BOOL
VAR_INPUT
END_VAR
IsDisassemblyCell := m_bIsDisassemblyCell;
END_METHOD

METHOD IsError : BOOL
VAR_INPUT
END_VAR
IF m_csCellState = CELL_STATE.e_ERROR THEN
	IsError := TRUE;
END_IF
END_METHOD

METHOD IsIdle : BOOL
VAR_INPUT
END_VAR
IF m_csCellState = CELL_STATE.e_IDEL THEN
	IsIdle := TRUE;
END_IF
END_METHOD

METHOD IsVirtualCell : BOOL
VAR_INPUT
END_VAR
IsVirtualCell :=FALSE;
END_METHOD

METHOD PUBLIC RequestActionState : BOOL
VAR_INPUT
	csStateRequest : CELL_ACTION_STATE;
END_VAR
m_csStateRequest := csStateRequest;
END_METHOD

METHOD RequestWork : BOOL
VAR_INPUT
END_VAR
m_csCellState := CELL_STATE.e_WORKING;
END_METHOD

METHOD SetDisassemblyCell : BOOL
VAR_INPUT
	bIsDisassemblyCell : BOOL;
END_VAR
m_bIsDisassemblyCell := bIsDisassemblyCell;
END_METHOD

METHOD SetGetDataServiceEnable : BOOL
VAR_INPUT
END_VAR
m_bDataServiceGetEnable := TRUE;
SetGetDataServiceEnable := TRUE;
END_METHOD

METHOD SetName : BOOL
VAR_INPUT
	sName :string ;
END_VAR
m_sName := sName;
END_METHOD

METHOD SetPutDataServiceEnable : BOOL
VAR_INPUT
END_VAR
m_bDataServicePutEnable := TRUE;
SetPutDataServiceEnable := TRUE;
END_METHOD

METHOD SetVirtualCell : BOOL
VAR_INPUT
END_VAR
END_METHOD

METHOD SetWorkpiece : BOOL
VAR_INPUT
	iWorkpiece : DINT;
	sWorkpieceID : STRING;
END_VAR
m_iWorkpiece := iWorkpiece;
m_sWorkpieceID := sWorkpieceID;
END_METHOD

METHOD PUBLIC StateMachine : BOOL
VAR_INPUT
END_VAR




fbInterface();
fbClamp();



// Error-Abfragen
IF fbClamp.IsError() THEN
	m_csCellState := CELL_STATE.e_ERROR; 
	m_sErrorString := 'CLAMP-Error: Clamp is closed without Workpiece';
END_IF


//Zellen Zustandsmaschine

CASE m_csCellState OF 
	CELL_STATE.e_IDEL:
		fbClamp.SetOpenClamp();	
	
		;
 	CELL_STATE.e_MHS_ACTION;
		//SubRoutine für Aktion beim beladen aktuell leer da alles vom MHS gesteuert wird 
	
		;
	CELL_STATE.e_WORKING:
		//SubRoutine zum Durchführen einer Bearbeitung
		
		IF NOT (m_csCellStateLast = m_csCellState) THEN
			m_csSRWorkingState := CELL_WORKING_STATES.e_START;
			IF m_bDataServiceGetEnable THEN
				fbDataServiceGet.SetNetIP('192.168.74.113.1.1');
				fbDataServiceGet.SetWorkingDirectory('C:\Users\Nübel\Desktop\Sysdem_Nü_Ulitmate\CUTS');
				m_sConfigString := 'C:\Users\Nübel\Desktop\Sysdem_Nü_Ulitmate\CUTS\';
				m_sConfigString := CONCAT(m_sConfigString , m_sName); // erstellen des Pfades der Applikation 
				m_sConfigString := CONCAT(m_sConfigString , m_sConfigStringEndGet);
				fbDataServiceGet.SetCommandLine(m_sWorkpieceID);
				fbDataServiceGet.SetPathOfApplication(m_sConfigString);
				fbDataServiceGet.StartDataService();
			END_IF
		END_IF
			
		CASE m_csSRWorkingState OF
			
			CELL_WORKING_STATES.e_START:
				
				IF NOT (m_csSRWorkingStateLast = m_csSRWorkingState )THEN
					m_csStateRequest := CELL_ACTION_STATE.e_Startabel;
				END_IF
				//m_csSRWorkingState:= CELL_WORKING_STATES.e_FINISHED;
				
				IF m_csState = CELL_ACTION_STATE.e_Startabel AND (fbDataServiceGet.IsFinished() OR NOT(m_bDataServiceGetEnable) )  THEN // Zelle bereit zum Starten und DataServiceGet fertig oder nicht konfiguriert
					m_csSRWorkingState:= CELL_WORKING_STATES.e_WORKING;
					fbDataServiceGet.SetIdle();
					m_csStateRequest:= CELL_ACTION_STATE.e_Running;
				END_IF
				
				
			CELL_WORKING_STATES.e_WORKING:
				IF NOT (m_csSRWorkingStateLast = m_csSRWorkingState) THEN
					m_csStateRequest := CELL_ACTION_STATE.e_Running;
				END_IF
				
				IF m_csState = CELL_ACTION_STATE.e_Finished THEN
					m_csSRWorkingState := CELL_WORKING_STATES.e_FINISHED;
					IF m_bDataServicePutEnable THEN
						fbDataServicePut.SetNetIP('192.168.74.113.1.1');
						fbDataServicePut.SetWorkingDirectory('C:\Users\Nübel\Desktop\Sysdem_Nü_Ulitmate\CUTS');
						m_sConfigString := 'C:\Users\Nübel\Desktop\Sysdem_Nü_Ulitmate\CUTS\';						
						m_sConfigString := CONCAT(m_sConfigString , m_sName); // erstellen des Pfades der Applikation 
						m_sConfigString := CONCAT(m_sConfigString , m_sConfigStringEndPut);// erstellen des Pfades der Applikation
						fbDataServicePut.SetCommandLine(m_sWorkpieceID);
						fbDataServicePut.SetPathOfApplication(m_sConfigString);
						fbDataServicePut.StartDataService();
						m_csSRWorkingState := e_DATAPUT;
					END_IF
		
				END_IF
			CELL_WORKING_STATES.e_DATAPUT:
				
					IF fbDataServicePut.IsFinished() THEN
						fbDataServicePut.SetIdle();
						m_csSRWorkingState := CELL_WORKING_STATES.e_FINISHED;
					END_IF
					
					IF fbDataServicePut.IsError() THEN
						fbDataServicePut.SetIdle();
						m_csSRWorkingState := CELL_STATE.e_ERROR;
					END_IF
					
			CELL_WORKING_STATES.e_FINISHED:
				m_csCellState := CELL_STATE.e_IDEL;
			
		END_CASE		
		
	CELL_STATE.e_ERROR:
		m_csState :=CELL_ACTION_STATE.e_ToEmergencyStop;
	
		
END_CASE
m_csSRWorkingStateLast := m_csSRWorkingState;
m_csCellStateLast := m_csCellState;

IF NOT (m_csStateRequestOld = m_csStateRequest) THEN
	m_csState := m_csStateRequest - 1;
	m_csStateRequestOld := m_csStateRequest;
END_IF


// Aktions Zustandsmaschine
CASE m_csState OF 
	CELL_ACTION_STATE.e_ToStandby:
		IF NOT (m_csStateLastCycle = m_csState) THEN
			fbInterface.SetStandby(TRUE);
			m_csStateLastAction := m_csStateLastCycle;
		END_IF
		
		IF fbInterface.GetStandby() THEN
			m_csState := e_Standby; 
		END_IF
		
	CELL_ACTION_STATE.e_Standby :
	
		IF NOT (m_csStateLastCycle = m_csState) THEN
			m_csStateLastAction := m_csStateLastCycle;
		END_IF
		fbInterface.SetStandby(FALSE);
		
	CELL_ACTION_STATE.e_ToLoadPos:
	
		IF NOT (m_csStateLastCycle = m_csState) THEN
			m_csStateLastAction := m_csStateLastCycle;
			fbInterface.SetMoveToLoad(TRUE);
			fbClamp.SetOpenClamp();
		END_IF
		
		IF fbInterface.GetLoadPos() AND fbClamp.IsOpen() THEN
			m_csState := e_LoadPos; 
		END_IF
		
		
	CELL_ACTION_STATE.e_LoadPos:
	
		IF NOT (m_csStateLastCycle = m_csState) THEN
			m_csStateLastAction := m_csStateLastCycle;
		END_IF
		fbInterface.SetMoveToLoad(FALSE);
				
		
	CELL_ACTION_STATE.e_ToStartabel:
	
		IF NOT (m_csStateLastCycle = m_csState) THEN
			m_csStateLastAction := m_csStateLastCycle;
			fbClamp.SetCloseClampFull();
		END_IF
		
		
		IF  fbClamp.IsClosedFull() THEN
			m_csState := e_Startabel; 
		END_IF
		
	CELL_ACTION_STATE.e_Startabel:
	
		IF NOT (m_csStateLastCycle = m_csState) THEN
			m_csStateLastAction := m_csStateLastCycle;
			
		END_IF
		
	CELL_ACTION_STATE.e_ToRunning:
	
		IF NOT (m_csStateLastCycle = m_csState) THEN
			m_csStateLastAction := m_csStateLastCycle;
			fbInterface.SetStart(TRUE);
		END_IF
		
		IF fbInterface.GetIsRunning() THEN
			m_csState := CELL_ACTION_STATE.e_Running; 
		END_IF
		
	CELL_ACTION_STATE.e_Running:
	
		IF NOT (m_csStateLastCycle = m_csState) THEN
			m_csStateLastAction := m_csStateLastCycle;
		END_IF
		fbInterface.SetStart(FALSE);
		IF fbInterface.GetFinished() THEN
			m_csState := CELL_ACTION_STATE.e_Finished;		
		END_IF
	CELL_ACTION_STATE.e_Finished:
		IF NOT (m_csStateLastCycle = m_csState) THEN
			m_csStateLastAction := m_csStateLastCycle;
		END_IF
		
	CELL_ACTION_STATE.e_ToUnLoadPos:
 
		IF NOT (m_csStateLastCycle = m_csState) THEN
			m_csStateLastAction := m_csStateLastCycle;
			fbClamp.SetOpenClamp();
			fbInterface.SetMoveToUnload(TRUE);
			
		END_IF
		
		
		IF fbInterface.GetUnloadPos() AND fbClamp.IsOpen() THEN
			m_csState := e_UnLoadPos; 
			fbInterface.SetMoveToUnload(FALSE);
		END_IF
		
	CELL_ACTION_STATE.e_UnLoadPos:
	
		IF NOT (m_csStateLastCycle = m_csState) THEN
			m_csStateLastAction := m_csStateLastCycle;
		END_IF
		
	CELL_ACTION_STATE.e_ToEmergencyStop:
	
		IF NOT (m_csStateLastCycle = m_csState) THEN
			m_csStateLastAction := m_csStateLastCycle;
		END_IF
		
		
		IF fbInterface.GetEmergencyStop() THEN
			m_csState := e_EmergencyStop; 
		END_IF
		
	CELL_ACTION_STATE.e_EmergencyStop:
	
		IF NOT (m_csStateLastCycle = m_csState) THEN
			m_csStateLastAction := m_csStateLastCycle;
		END_IF
		
	CELL_ACTION_STATE.e_ToEmergencyOff:
	
		IF NOT (m_csStateLastCycle = m_csState) THEN
			m_csStateLastAction := m_csStateLastCycle;
		END_IF
		
		
		IF fbInterface.GetEmergencyStop() THEN
			m_csState := e_EmergencyOff; 
		END_IF
		
	CELL_ACTION_STATE.e_EmergencyOff:
	
		IF NOT (m_csStateLastCycle = m_csState) THEN
			m_csStateLastAction := m_csStateLastCycle;
		END_IF
		
	ELSE
		IF NOT (m_csStateLastCycle = m_csState) THEN
			m_csStateLastAction := m_csStateLastCycle;
		END_IF
		
END_CASE

IF m_bDataServiceGetEnable THEN
	fbDataServiceGet();
END_IF
IF m_bDataServicePutEnable THEN	
	fbDataServicePut();
END_IF

m_csStateLastCycle := m_csState;
END_METHOD

METHOD StateMachineProfibus : BOOL
//*Hami* zum Anschluss an Profibus vorgesehen 
//*Hami* Moentan nur bei LaseTec Aktiviert ist
//*Hami* bei andere Zelle ist inaktiv 
//*Hami* bei andere Zelle ist StateMachine Aktiv
VAR_INPUT
END_VAR
//////////////////////////////////////////////////////////////////////////////////////////////////////
//*Hami* Aufruf von FB_InterfaceProfibus zur Ausführung
//*Hami* In Method(StateMachine) wird FB_InterfaceIO aufgerufen (einziger Unterschied Zwischen StateMachineProfibus und StateMachine)
fbInterfaceProfibus();
//////////////////////////////////////////////////////////////////////////////////////////////////////

fbClamp();



// Error-Abfragen
IF fbClamp.IsError() THEN
	m_csCellState := CELL_STATE.e_ERROR; 
	m_sErrorString := 'CLAMP-Error: Clamp is closed without Workpiece';
END_IF


//Zellen Zustandsmaschine

CASE m_csCellState OF 
	CELL_STATE.e_IDEL:
		fbClamp.SetOpenClamp();	
	
		;
 	CELL_STATE.e_MHS_ACTION;
		//SubRoutine für Aktion beim beladen aktuell leer da alles vom MHS gesteuert wird 
	
		;
	CELL_STATE.e_WORKING:
		//SubRoutine zum Durchführen einer Bearbeitung
		
		IF NOT (m_csCellStateLast = m_csCellState) THEN
			m_csSRWorkingState := CELL_WORKING_STATES.e_START;
			IF m_bDataServiceGetEnable THEN
				fbDataServiceGet.SetNetIP('192.168.74.113.1.1');
				fbDataServiceGet.SetWorkingDirectory('C:\Users\Nübel\Desktop\Sysdem_Nü_Ulitmate\CUTS');
				m_sConfigString := 'C:\Users\Nübel\Desktop\Sysdem_Nü_Ulitmate\CUTS\';
				m_sConfigString := CONCAT(m_sConfigString , m_sName); // erstellen des Pfades der Applikation 
				m_sConfigString := CONCAT(m_sConfigString , m_sConfigStringEndGet);
				fbDataServiceGet.SetCommandLine(m_sWorkpieceID);
				fbDataServiceGet.SetPathOfApplication(m_sConfigString);
				fbDataServiceGet.StartDataService();
			END_IF
		END_IF
			
		CASE m_csSRWorkingState OF
			
			CELL_WORKING_STATES.e_START:
				
				IF NOT (m_csSRWorkingStateLast = m_csSRWorkingState )THEN
					m_csStateRequest := CELL_ACTION_STATE.e_Startabel;
				END_IF
				//m_csSRWorkingState:= CELL_WORKING_STATES.e_FINISHED;
				
				IF m_csState = CELL_ACTION_STATE.e_Startabel AND (fbDataServiceGet.IsFinished() OR NOT(m_bDataServiceGetEnable) )  THEN // Zelle bereit zum Starten und DataServiceGet fertig oder nicht konfiguriert
					m_csSRWorkingState:= CELL_WORKING_STATES.e_WORKING;
					fbDataServiceGet.SetIdle();
					m_csStateRequest:= CELL_ACTION_STATE.e_Running;
				END_IF
				
				
			CELL_WORKING_STATES.e_WORKING:
				IF NOT (m_csSRWorkingStateLast = m_csSRWorkingState) THEN
					m_csStateRequest := CELL_ACTION_STATE.e_Running;
				END_IF
				
				IF m_csState = CELL_ACTION_STATE.e_Finished THEN
					m_csSRWorkingState := CELL_WORKING_STATES.e_FINISHED;
					IF m_bDataServicePutEnable THEN
						fbDataServicePut.SetNetIP('192.168.74.113.1.1');
						fbDataServicePut.SetWorkingDirectory('C:\Users\Nübel\Desktop\Sysdem_Nü_Ulitmate\CUTS');
						m_sConfigString := 'C:\Users\Nübel\Desktop\Sysdem_Nü_Ulitmate\CUTS\';						
						m_sConfigString := CONCAT(m_sConfigString , m_sName); // erstellen des Pfades der Applikation 
						m_sConfigString := CONCAT(m_sConfigString , m_sConfigStringEndPut);// erstellen des Pfades der Applikation
						fbDataServicePut.SetCommandLine(m_sWorkpieceID);
						fbDataServicePut.SetPathOfApplication(m_sConfigString);
						fbDataServicePut.StartDataService();
						m_csSRWorkingState := e_DATAPUT;
					END_IF
		
				END_IF
			CELL_WORKING_STATES.e_DATAPUT:
				
					IF fbDataServicePut.IsFinished() THEN
						fbDataServicePut.SetIdle();
						m_csSRWorkingState := CELL_WORKING_STATES.e_FINISHED;
					END_IF
					
					IF fbDataServicePut.IsError() THEN
						fbDataServicePut.SetIdle();
						m_csSRWorkingState := CELL_STATE.e_ERROR;
					END_IF
					
			CELL_WORKING_STATES.e_FINISHED:
				m_csCellState := CELL_STATE.e_IDEL;
			
		END_CASE		
		
	CELL_STATE.e_ERROR:
		m_csState :=CELL_ACTION_STATE.e_ToEmergencyStop;
	
		
END_CASE
m_csSRWorkingStateLast := m_csSRWorkingState;
m_csCellStateLast := m_csCellState;

IF NOT (m_csStateRequestOld = m_csStateRequest) THEN
	m_csState := m_csStateRequest - 1;
	m_csStateRequestOld := m_csStateRequest;
END_IF


// Aktions Zustandsmaschine
CASE m_csState OF 
	CELL_ACTION_STATE.e_ToStandby:
		IF NOT (m_csStateLastCycle = m_csState) THEN
			fbInterface.SetStandby(TRUE);
			m_csStateLastAction := m_csStateLastCycle;
		END_IF
		
		IF fbInterface.GetStandby() THEN
			m_csState := e_Standby; 
		END_IF
		
	CELL_ACTION_STATE.e_Standby :
	
		IF NOT (m_csStateLastCycle = m_csState) THEN
			m_csStateLastAction := m_csStateLastCycle;
		END_IF
		fbInterface.SetStandby(FALSE);
		
	CELL_ACTION_STATE.e_ToLoadPos:
	
		IF NOT (m_csStateLastCycle = m_csState) THEN
			m_csStateLastAction := m_csStateLastCycle;
			fbInterface.SetMoveToLoad(TRUE);
			fbClamp.SetOpenClamp();
		END_IF
		
		IF fbInterface.GetLoadPos() AND fbClamp.IsOpen() THEN
			m_csState := e_LoadPos; 
		END_IF
		
		
	CELL_ACTION_STATE.e_LoadPos:
	
		IF NOT (m_csStateLastCycle = m_csState) THEN
			m_csStateLastAction := m_csStateLastCycle;
		END_IF
		fbInterface.SetMoveToLoad(FALSE);
				
		
	CELL_ACTION_STATE.e_ToStartabel:
	
		IF NOT (m_csStateLastCycle = m_csState) THEN
			m_csStateLastAction := m_csStateLastCycle;
			fbClamp.SetCloseClampFull();
		END_IF
		
		
		IF  fbClamp.IsClosedFull() THEN
			m_csState := e_Startabel; 
		END_IF
		
	CELL_ACTION_STATE.e_Startabel:
	
		IF NOT (m_csStateLastCycle = m_csState) THEN
			m_csStateLastAction := m_csStateLastCycle;
			
		END_IF
		
	CELL_ACTION_STATE.e_ToRunning:
	
		IF NOT (m_csStateLastCycle = m_csState) THEN
			m_csStateLastAction := m_csStateLastCycle;
			fbInterface.SetStart(TRUE);
		END_IF
		
		IF fbInterface.GetIsRunning() THEN
			m_csState := CELL_ACTION_STATE.e_Running; 
		END_IF
		
	CELL_ACTION_STATE.e_Running:
	
		IF NOT (m_csStateLastCycle = m_csState) THEN
			m_csStateLastAction := m_csStateLastCycle;
		END_IF
		fbInterface.SetStart(FALSE);
		IF fbInterface.GetFinished() THEN
			m_csState := CELL_ACTION_STATE.e_Finished;		
		END_IF
	CELL_ACTION_STATE.e_Finished:
		IF NOT (m_csStateLastCycle = m_csState) THEN
			m_csStateLastAction := m_csStateLastCycle;
		END_IF
		
	CELL_ACTION_STATE.e_ToUnLoadPos:
 
		IF NOT (m_csStateLastCycle = m_csState) THEN
			m_csStateLastAction := m_csStateLastCycle;
			fbClamp.SetOpenClamp();
			fbInterface.SetMoveToUnload(TRUE);
			
		END_IF
		
		
		IF fbInterface.GetUnloadPos() AND fbClamp.IsOpen() THEN
			m_csState := e_UnLoadPos; 
			fbInterface.SetMoveToUnload(FALSE);
		END_IF
		
	CELL_ACTION_STATE.e_UnLoadPos:
	
		IF NOT (m_csStateLastCycle = m_csState) THEN
			m_csStateLastAction := m_csStateLastCycle;
		END_IF
		
	CELL_ACTION_STATE.e_ToEmergencyStop:
	
		IF NOT (m_csStateLastCycle = m_csState) THEN
			m_csStateLastAction := m_csStateLastCycle;
		END_IF
		
		
		IF fbInterface.GetEmergencyStop() THEN
			m_csState := e_EmergencyStop; 
		END_IF
		
	CELL_ACTION_STATE.e_EmergencyStop:
	
		IF NOT (m_csStateLastCycle = m_csState) THEN
			m_csStateLastAction := m_csStateLastCycle;
		END_IF
		
	CELL_ACTION_STATE.e_ToEmergencyOff:
	
		IF NOT (m_csStateLastCycle = m_csState) THEN
			m_csStateLastAction := m_csStateLastCycle;
		END_IF
		
		
		IF fbInterface.GetEmergencyStop() THEN
			m_csState := e_EmergencyOff; 
		END_IF
		
	CELL_ACTION_STATE.e_EmergencyOff:
	
		IF NOT (m_csStateLastCycle = m_csState) THEN
			m_csStateLastAction := m_csStateLastCycle;
		END_IF
		
	ELSE
		IF NOT (m_csStateLastCycle = m_csState) THEN
			m_csStateLastAction := m_csStateLastCycle;
		END_IF
		
END_CASE

IF m_bDataServiceGetEnable THEN
	fbDataServiceGet();
END_IF
IF m_bDataServicePutEnable THEN	
	fbDataServicePut();
END_IF

m_csStateLastCycle := m_csState;
END_METHOD

END_FUNCTION_BLOCK

// ---- POUs/FB_ClampSimulated.TcPOU
FUNCTION_BLOCK FB_ClampSimulated
VAR_INPUT
	
END_VAR
VAR_OUTPUT
END_VAR
VAR
m_csState : CLAMP_STATE;	
m_csStateRequested : CLAMP_STATE;

//Eingänge
m_bIsOpen : BOOL;
m_bIsClosed : BOOL;
m_bIsClosedFull : BOOL;

//Ausgänge
m_bOpen :BOOL;
m_bClose :BOOL;

iWaitingTime : INT := 500;
iTimer: INT := 0;

END_VAR


StateMachine();

METHOD IsClosed : BOOL
VAR_INPUT
END_VAR

VAR
END_VAR
iTimer := iTimer +1;

IF iTimer > iWaitingTime THEN
	m_bIsClosed := TRUE;
	iTimer := 0;	
END_IF

IF m_csState = CLAMP_STATE.e_CLOSED THEN
	IsClosed := TRUE;
END_IF
END_METHOD

METHOD IsClosedFull : BOOL
VAR_INPUT
END_VAR

VAR
END_VAR

iTimer := iTimer +1;

IF iTimer > iWaitingTime THEN
	m_bIsClosedFull := TRUE;
	iTimer := 0;	
END_IF

IF m_csState = CLAMP_STATE.e_CLOSED_FULL THEN
	IsClosedFull := TRUE;
END_IF
END_METHOD

METHOD IsError : BOOL
VAR_INPUT
END_VAR
IF m_csState = CLAMP_STATE.e_ERROR THEN
	IsError := TRUE;
END_IF
END_METHOD

METHOD IsOpen : BOOL
VAR_INPUT
END_VAR

VAR
END_VAR
iTimer := iTimer +1;

IF iTimer > iWaitingTime THEN
	m_bIsOpen := TRUE;
	iTimer := 0;	
END_IF

IF m_csState = CLAMP_STATE.e_OPEN THEN
	IsOpen := TRUE;
END_IF
END_METHOD

METHOD SetCloseClampEmpty : BOOL
VAR_INPUT
END_VAR
m_csStateRequested := CLAMP_STATE.e_CLOSED;
m_bClose := TRUE;
SetCloseClampEmpty:=TRUE;
END_METHOD

METHOD SetCloseClampFull : BOOL
VAR_INPUT
END_VAR
m_csStateRequested := CLAMP_STATE.e_CLOSED_FULL;
m_bClose := TRUE;
SetCloseClampFull := TRUE;
END_METHOD

METHOD SetOpenClamp : BOOL
VAR_INPUT
END_VAR
m_bOpen := TRUE;
END_METHOD

METHOD StateMachine : BOOL
VAR_INPUT
END_VAR

//m_bIsOpen : BOOL;
//m_bIsClosed : BOOL;
//m_bIsClosedFull : BOOL;

CASE m_csState  OF
	
	CLAMP_STATE.e_OPEN:	
		

		IF m_bIsClosed THEN
			m_csState := CLAMP_STATE.e_CLOSED;		
		END_IF
		
		IF m_bIsClosedFull THEN
			m_csState := CLAMP_STATE.e_CLOSED_FULL;		
		END_IF
		
 	CLAMP_STATE.e_CLOSED_FULL:
	// Fehler wenn falscher Zustand
 		IF m_csStateRequested = CLAMP_STATE.e_CLOSED THEN
  			m_csState := CLAMP_STATE.e_ERROR;
		END_IF
		
		
		IF m_bIsOpen THEN
			m_csState := CLAMP_STATE.e_OPEN;		
		END_IF
	
	CLAMP_STATE.e_CLOSED:
			// Fehler wenn falscher Zustand in diesem Fall: Werkstück erwartet aber nicht im Halter
 		IF m_csStateRequested = CLAMP_STATE.e_CLOSED_FULL THEN
  			m_csState := CLAMP_STATE.e_ERROR;
		END_IF
	
	
		IF m_bIsOpen THEN
			m_csState := CLAMP_STATE.e_OPEN;		
		END_IF
		
CLAMP_STATE.e_ERROR:
		
END_CASE
END_METHOD

END_FUNCTION_BLOCK

// ---- POUs/MAIN.TcPOU

PROGRAM MAIN
	
VAR



// Allg. nitwendige Variablen
m_bInit : BOOL;
I : DINT;
sString : STRING;
diDint : DINT;
bBOOL:BOOL;
m_iCellUpdateIter : INT := 0; // Iterationsvariable für die Json Strings der Zelle

// Zellen //NN
fbCellA2 : FB_Cell;
fbCellA5 : FB_Cell; 
///////////////////////////////////////////////////////////////////////////////////////////////////////
fbCellL1 : FB_Cell;   //*Hami*  Deklaration ein neues FB_Cell für LaserTec
///////////////////////////////////////////////////////////////////////////////////////////////////////
fbCellD1 : FB_Cell_Simu;  //Ist eine andere Zelle, kann mann einzeln ändern
fbCellV1 : FB_VirtualCell;
//fbCellV2 : FB_VirtualCell;

//An die Anzahl der Zellen anpassen
///////////////////////////////////////////////////////////////////////////////////////////////////////
//*Hami* Anzahl von Zellen auf 5 einstellen + LaserTec
//////////////////////////////////////////////////////////////////////////////////////////////////////
aCellList : ARRAY [1..5] OF I_CELL; // Liste der Zellen //NN
m_iNumberOfCells : DINT := 4; // Bei hinzufügen/löschen einer Zelle ist hier die Anzahl anzupassen  //NN

// MHS 
fbMHS : FB_MHS;
//fb_put : FB_TestHTTP_HeaderAuth ; 

// Kommunikations-Variabeln für Aktionen von der GUI


m_bTrigger : BOOL;// Trigger zum zyklischen Aktualisieren der Anwendung
m_iTriggerTimer : INT; // Zähler zum Trigger 
m_sJsonTrigger : STRING(80);

m_sActionID : STRING(80);
m_sWPID : STRING(80);
m_iWPRequest : DINT;
m_sCellRequest : STRING;
m_iActionRequest : DINT;
m_iActionState : DINT;


m_sActionIDLast : STRING(80);
m_sWPIDLast : STRING(80);
m_iWPRequestLast : DINT;
m_iCellRequestLast : DINT;
m_iActionRequestLast : DINT;
m_iActionStateLast : DINT;
m_iCellRequest : DINT;

m_bAktionInProgress : BOOL; 

//JSON-Variablen
	//Writer
	m_iJsonTimer 		: DINT;
 	dtTimestamp 		: DATE_AND_TIME := DT#2017-04-04-12:42:42;
 	fbJson      		: FB_JsonSaxWriter;
 	sJsonDocCells   	: STRING(3000);
	//Reader
 	fbJsonReader    		: FB_JsonSaxReader;
	pJsonParse 				: JsonSaxHandler;
	sJsonDocAction			: STRING(255);
	sJsonDocLastAction   : STRING(255);
	
	sJsonDocError 		 : STRING (255); 

END_VAR


//Initialisierung
IF NOT m_bInit THEN
	// Hier die FunktionsBlöcke der Maschinen in das Array Schreiben !!! //NN
	aCellList[1] := fbCellA2;
	aCellList[1].SetName('A2'); // Geometrieerfassung
	aCellList[1].SetGetDataServiceEnable();

	aCellList[2] := fbCellD1;
	aCellList[2].SetName('D1'); // LaserSchweißen
	//aCellList[2].SetGetDataServiceEnable();  //Liest in den Zwilling aus
	//aCellList[2].SetPutDataServiceEnable();   //Schreibt in den Zwilling rein
	
	//Array an die Anzahl der Zellen anpassen
	aCellList[3] := fbCellA5;
	aCellList[3].SetName('A5'); // Demontage
	
	aCellList[4] := fbCellV1;
	aCellList[4].SetName('V1'); 		// Virtuell
	aCellList[4].SetVirtualCell();		//Ist eine Virtuelle zelle
	
///////////////////////////////////////////////////////////////////////////////////////////////////////	
	aCellList[5] := fbCellL1;			//*Hami*  FB für LaserTec 
	aCellList[5].SetName('L1');
///////////////////////////////////////////////////////////////////////////////////////////////////////

	// Intitialisiert setzen 
	m_bInit := TRUE;

END_IF



IF m_bAktionInProgress = FALSE THEN 
	// Abfrage ob neue Aktion angestoßen wurde
	CheckForNewAction();
		
END_IF


//Zustandmaschinen
	// Zyklische aktualisierung der Zellen-Zustandsmaschinen
	I := 1;
	FOR I:=1 TO m_iNumberOfCells BY 1 DO
    	aCellList[I].StateMachine();
	END_FOR;
///////////////////////////////////////////////////////////////////////////////////////////////////////	
	//*Hami* Zyklische aktualisierung der Lasertec-Zustandsmaschinen mit Profibus
	aCellList[5].StateMachineProfibus();
///////////////////////////////////////////////////////////////////////////////////////////////////////	
	// Zyklische aktualisierung der MHS-Zustandsmaschine
	fbMHS();
// Zustandsmaschinen durchgelaufen

IF m_bAktionInProgress THEN// MHS muss den Zustand der involvierten Zelle kennen und eine Zustand von der Zelle anfordern können
	
	fbMHS.SetStateCurrentMachineForAction( aCellList[fbMHS.GetCurrentCellForAction()].GetState());// Aktualisieren des MHS Zustandes
	IF fbMHS.NeededCellStatePending() THEN // Wenn das MHS einen Zellenzustand verlangt wird er folgend übergeben
		aCellList[fbMHS.GetCurrentCellForAction()].RequestActionState(fbMHS.SendNeededToCell() );// Übergabe des geforderten Zellenzustandes an die Zelle
	END_IF
END_IF


// Abfrage ob letzte Aktion Abgeschlossen wurde.... auf WIN abgefragen um neue Aktion zu senden 
IF fbMHS.GetActionFinished() THEN
	m_bAktionInProgress := FALSE; 
	IF m_iActionRequestLast = 2 THEN // Bestuecken
		aCellList[m_iCellRequestLast].SetWorkpiece(m_iWPRequestLast, m_sWPIDLast);// Werkstück an die Zelle übergeben
		aCellList[m_iCellRequestLast].RequestWork(); // Starten der Bearbeitung in der Zelle		
	ELSE
		aCellList[m_iCellRequestLast].SetWorkpiece(0, 'Empty'); // Werkstück der Zelle nehmen
	END_IF
	m_iActionStateLast := 3;
END_IF

// Schreiben der JSON-Strings zur Kommunikation der Systemdemostrator-Anwendung
WriteJsonStrings();

METHOD CheckForNewAction : BOOL
VAR_INPUT
END_VAR
	 ParseNewAction();
	m_iCellRequest := NumberOfCellName(m_sCellRequest);
	IF	 (NOT(m_sActionID = m_sActionIDLast)) AND (m_iCellRequest <= m_iNumberOfCells) AND (m_iCellRequest > 0) THEN // Neue Aktion und Zelle ist existent
		IF NOT(aCellList[m_iCellRequest].IsVirtualCell())THEN
			
			IF aCellList[m_iCellRequest].IsIdle() THEN // Zelle frei
				// Neue Aktion an das MHS übergeben 
				WriteNewActionToMHS();
				m_bAktionInProgress := TRUE;// Setzen des Flags 
			END_IF
		ELSE // Im Falle einer Aktion für eine virtuelle Zelle
			IF aCellList[m_iCellRequest].IsIdle() THEN
				aCellList[m_iCellRequest].SetWorkpiece(0, m_sWPID );
				aCellList[m_iCellRequest].RequestWork();	
				//m_iActionStateLast := 3; // Wird nur angestoßen ist direkt fertig mit der Aktion, so dass eine weitere beginnen kann.
			END_IF
		END_IF
	
	END_IF
END_METHOD

METHOD NumberOfCellName : DINT
VAR_INPUT
	sNameOfCell : STRING;
END_VAR
FOR I:=1 TO m_iNumberOfCells BY 1 DO
    IF sNameOfCell = aCellList[I].GetName() THEN
		NumberOfCellName :=I;
	END_IF
END_FOR;
END_METHOD

METHOD ParseNewAction : BOOL
VAR_INPUT
END_VAR

	// Aktion JSonDoc Lesen des Aktuellen Strings
	fbJsonReader.Parse( sJson := sJsonDocAction, ipHdl := pJsonParse);
	
	IF pJsonParse.IsFinished() THEN
		// Übergabe der geparsten Variablen
		m_sActionID	:=	pJsonParse.GetActionID();
		m_sWPID	:=	pJsonParse.GetWPID();
		m_iWPRequest := pJsonParse.GetWPPlace(); 
		m_sCellRequest := pJsonParse.GetCell(); 
		m_iActionRequest:=pJsonParse.GetActionType();
		
		// Für den nächsten Durchlauf zurücksetzen 
		pJsonParse.Reset();
	ELSE
		// Parsen des Json-Strings
		fbJsonReader.Parse( sJson := sJsonDocAction, ipHdl := pJsonParse);
	END_IF
END_METHOD

METHOD WriteJSonDocAction : BOOL
VAR_INPUT
END_VAR

fbJson.ResetDocument();
		//fbJson.StartArray();
fbJson.StartObject();
            fbJson.AddKey('m_sActionID');
			fbJson.AddString(m_sActionIDLast);
            fbJson.AddKey('m_sWPID');
			sString := m_sWPIDLast;
			fbJson.AddString(sString);
            fbJson.AddKey('m_iWPPlace');
			fbJson.AddDint(m_iWPRequestLast);
            fbJson.AddKey('m_sCell');
			IF m_iCellRequestLast > 0 THEN// Sonst würden das Zell Array außerhalb seines Bereiches angesproehcen werden
				sString := aCellList[m_iCellRequestLast].GetName();
			ELSE
				sString := 'EmptyAction';				
			END_IF
			fbJson.AddString(sString);
            fbJson.AddKey('m_eActionType');
			fbJson.AddDint(m_iActionRequestLast);
            fbJson.AddKey('m_iActionState');
			fbJson.AddDint(m_iActionStateLast);	
fbJson.EndObject();
	sJsonDocLastAction := fbJson.GetDocument();

WriteJSonDocAction := TRUE;
END_METHOD

METHOD WriteJSonDocCells : BOOL
VAR_INPUT
END_VAR
// Merken alle Zellen einzelnd Updaten, weil es nicht möglich ist die über 255 Zeichen langen Strings aller zu übertragen

	fbJson.ResetDocument();
	//fbJson.StartObject();
	//fbJson.AddKey('Timestamp');
	
	//fbJson.AddDateTime(dtTimestamp);
	m_iCellUpdateIter := m_iCellUpdateIter +1 ; 
	IF m_iCellUpdateIter > m_iNumberOfCells THEN
		m_iCellUpdateIter := 1;
	END_IF
		//fbJson.AddKey('Cell');
		m_sActionIDLast := m_sActionID;
		m_iWPRequestLast := m_iWPRequest; 		
		m_iCellRequestLast := m_iCellRequest;
		m_iActionRequestLast :=	m_iActionRequest;
		fbJson.StartObject();
		//fbJson.StartArray();
		fbJson.AddKey('Name');
		sString := aCellList[m_iCellUpdateIter].GetName();
		fbJson.AddString(sString);
		fbJson.AddKey('State');
		fbJson.AddDint(aCellList[m_iCellUpdateIter].GetState());
		fbJson.AddKeyBool('Idle',aCellList[m_iCellUpdateIter].IsIdle());
		fbJson.AddKey('Workpiece');
		fbJson.AddDint(aCellList[m_iCellUpdateIter].GetWorkpiece());
		fbJson.AddKey('IsDisassemblyCell');
		fbJson.AddBool(aCellList[m_iCellUpdateIter].IsDisassemblyCell());
		fbJson.AddKey('IsVirtualCell');
		fbJson.AddBool(aCellList[m_iCellUpdateIter].IsVirtualCell());
		fbJson.EndObject();
		
		

	
	
	//fbJson.EndObject();
	sJsonDocCells := '';
	sJsonDocCells := fbJson.GetDocument();
	
WriteJSonDocCells := TRUE;
END_METHOD

METHOD WriteJSonError : BOOL
VAR_INPUT
END_VAR
	fbJson.ResetDocument();


	I := 1;
	FOR I:=1 TO m_iNumberOfCells BY 1 DO
		IF aCellList[I].IsError() THEN
			fbJson.StartObject();
			fbJson.AddKey('Name');
			sString := aCellList[I].GetName();
			fbJson.AddString(sString);	
			fbJson.AddKey('Workpiece');
			fbJson.AddDint(aCellList[I].GetWorkpiece());
			fbJson.AddKey('Error');
			sString := aCellList[I].GetErrorString();
			fbJson.AddString(sString);
			fbJson.EndObject();	
			
			sJsonDocError := '';
			sJsonDocError := fbJson.GetDocument();

		END_IF	
	
	END_FOR;
END_METHOD

METHOD WriteJsonStrings : BOOL
VAR_INPUT
END_VAR




// Erstellen eines Json-Strings für die GUI alle 100 Durchläufe 0,1s
m_iJsonTimer := m_iJsonTimer+1;
IF m_iJsonTimer > 150 THEN
	WriteJSonDocCells();
	WriteJSonDocAction();
	
	m_iJsonTimer := 0;
	
END_IF
// GUI Trigger um zyklische Aufrufe auch bei nicht veränderten JSON-Strings zu erzielen
// Ohne den Trigger würde ine Prüfung des Regenerationspfades bei nicht mehr vorhanden Aktion im Pfad nicht fortgeführt werden
IF m_iTriggerTimer > 2500 THEN
	m_bTrigger :=  NOT(m_bTrigger);// Bool abwechselnd false und true
	WriteJsonTrigger();
	m_iTriggerTimer := 0; 
END_IF
	
m_iTriggerTimer := m_iTriggerTimer + 1;
END_METHOD

METHOD WriteJsonTrigger : BOOL
VAR_INPUT
END_VAR
fbJson.ResetDocument();
		//fbJson.StartArray();
fbJson.StartObject();
            fbJson.AddKey('m_bTrigger');
			fbJson.AddBool(m_bTrigger);
fbJson.EndObject();
	m_sJsonTrigger := fbJson.GetDocument();
END_METHOD

METHOD WriteNewActionToMHS : BOOL
VAR_INPUT
END_VAR
// Übergaben der neuen Aktion an das MHS
fbMHS.RequestAction(	iWorkpiece := m_iWPRequest, iCell := m_iCellRequest, bRequest := m_iActionRequest);
// Speichern des Zustandes
m_sActionIDLast := m_sActionID;
m_sWPIDLast := m_sWPID; 
m_iWPRequestLast := m_iWPRequest; 		
m_iCellRequestLast := m_iCellRequest;
m_iActionRequestLast :=	m_iActionRequest;

m_iActionStateLast := 2;
END_METHOD

END_PROGRAM
